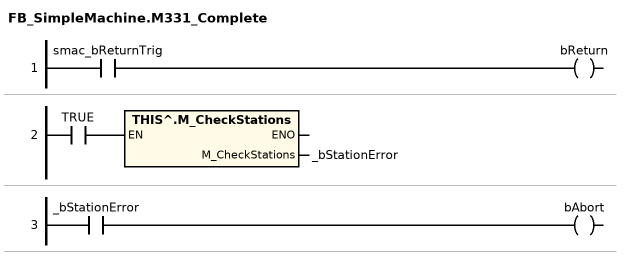
// NETWORK 1
bReturn := smac_bReturnTrig;

// NETWORK 2
_bStationError := THIS^.M_CheckStations();

// NETWORK 3
bAbort := _bStationError;
END_METHOD

(* In this state the most recent execution status should be maintained while
awaiting an explicit 'Unhold' command once internal conditions are satisfactory. *)
METHOD M411_Held : BOOL
VAR_OUTPUT
	(* This should be set to true if an explicit 'Unhold' command is received.
	Once set to true, the state machine will move to the 'Unholding' state. *)
	bUnhold	: BOOL;
	(* This should be set to true if an external source requests that the module
	exit its current state and come to a controlled stop. Once set to true, the
	state machine will move to the 'Stopping' state. *)
	bStop	: BOOL;
	(* This should be set to true if a potentially hazardous error or a safety
	fault has occurred in any tasks. Once set to true, the state machine will
	move to the 'Aborting' state. *)
	bAbort	: BOOL;
END_VAR
VAR
	_bStationError: BOOL;
END_VAR
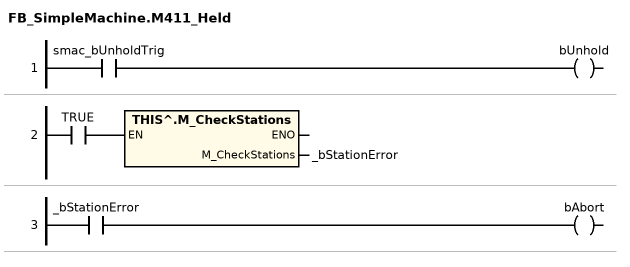
// NETWORK 1
bUnhold := smac_bUnholdTrig;

// NETWORK 2
_bStationError := THIS^.M_CheckStations();

// NETWORK 3
bAbort := _bStationError;
END_METHOD

(* In this state the most recent execution status should be maintained while
awaiting an explicit 'Unsuspend' command once external conditions are satisfactory. *)
METHOD M511_Suspended : BOOL
VAR_OUTPUT
	(* This should be set to true if an explicit 'Unsuspend' command is received.
	Once set to true, the state machine will move to the 'Unsuspending' state. *)
	bUnsuspend	: BOOL;
	(* This should be set to true if an external source requests that the module
	exit its current state and come to a controlled stop. Once set to true, the
	state machine will move to the 'Stopping' state. *)
	bStop	: BOOL;
	(* This should be set to true if a potentially hazardous error or a safety
	fault has occurred in any tasks. Once set to true, the state machine will
	move to the 'Aborting' state. *)
	bAbort	: BOOL;
END_VAR
VAR
	_bStationError: BOOL;
END_VAR
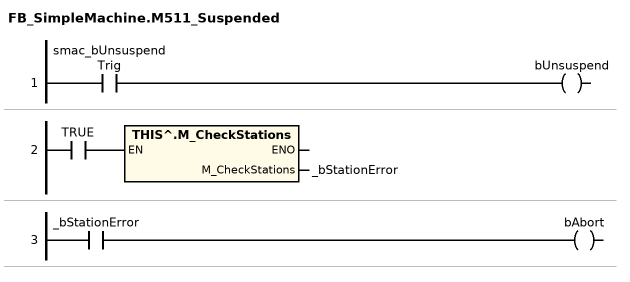
// NETWORK 1
bUnsuspend := smac_bUnsuspendTrig;

// NETWORK 2
_bStationError := THIS^.M_CheckStations();

// NETWORK 3
bAbort := _bStationError;
END_METHOD

END_FUNCTION_BLOCK

// Concrete/FB_StandardStation
FUNCTION_BLOCK FB_StandardStation EXTENDS FB_Station
VAR CONSTANT
	intMAX_USER_PROMPTS: INT := 255;
END_VAR
VAR_INPUT
	(* Station will start running process cycle once this is set to
		TRUE, and then will wait for this to be set to FALSE before
		resetting back to initial step. *)
	in_bRunCycleCommand: BOOL;
	(* Array of user prompts. *)
	in_arrUserPrompts: ARRAY[1..255] OF ST_Prompt;
	(* User retry signal for an exception state. *)
	in_bUserRetry: BOOL;
	(* User stop machine signal for an exception state. *)
	in_bUserAbort: BOOL;
END_VAR
VAR_OUTPUT
	(* Station should set this to TRUE while the process cycle is
		not running, and FALSE while running. *)
	out_bReadyToRun: BOOL;
	(* ID of the current user prompt. *)
	out_udintUserPromptCode: UDINT;
	(* Default message of the current user prompt. *)
	out_strUserPromptMessage: T_MaxString;
END_VAR
VAR
END_VAR

(* Sets ready to run to TRUE and waits for run cycle command to be reset. *)
METHOD M_AwaitCycleEnd : BOOL
VAR_INPUT
END_VAR
M_AwaitCycleEnd := FALSE;
IF NOT out_bReadyToRun THEN
	THIS^.M_LogMessage('Cycle complete.');
END_IF
out_bReadyToRun := TRUE;
IF NOT in_bRunCycleCommand THEN
	M_AwaitCycleEnd := TRUE;
END_IF
END_METHOD

(* Sets ready to run to TRUE and then waits for run cycle command. *)
METHOD M_AwaitCycleStart : BOOL
VAR_INPUT
END_VAR
M_AwaitCycleStart := FALSE;
out_bReadyToRun := TRUE;
IF in_bRunCycleCommand THEN
	out_bReadyToRun := FALSE;
	M_AwaitCycleStart := TRUE;
END_IF
END_METHOD

(* Clears the user prompt outputs. *)
METHOD M_ClearUserPrompt : BOOL
VAR_INPUT
END_VAR
out_strUserPromptMessage := '';
out_udintUserPromptCode := 0;
M_ClearUserPrompt := TRUE;
END_METHOD

(* Sets user prompt based on given code, and awaits user input. *)
METHOD M_HandleException : BOOL
VAR_INPUT
	(* Prompt code for the exception message. *)
	_in_udintPromptCode: UDINT;
	(* Error code to set in case user aborts. *)
	_in_udintErrorCode: UDINT;
END_VAR
VAR_OUTPUT
END_VAR
M_HandleException := FALSE;
THIS^.M_SetUserPrompt(_in_udintPromptCode);
IF in_bUserRetry THEN
	THIS^.M_ClearUserPrompt();
	M_HandleException := TRUE;
ELSIF in_bUserAbort THEN
	THIS^.M_SetError(_in_udintErrorCode, 'User chose to abort after an exception.');
END_IF
END_METHOD

METHOD M_ResetCycle : BOOL
VAR_INPUT
END_VAR
out_bReadyToRun := FALSE;
M_ResetCycle := TRUE;
END_METHOD

(* Sets out_strUserPromptCode and out_strUserPromptMessage based on
	the given user prompt code. *)
METHOD M_SetUserPrompt : BOOL
VAR_INPUT
	(* Prompt code to use for this user prompt. *)
	_in_udintCode: UDINT;
END_VAR

VAR
	_strMessage: T_MaxString;
	_intIndex: INT;
END_VAR
FOR _intIndex := 1 TO intMAX_USER_PROMPTS DO
	IF in_arrUserPrompts[_intIndex].udintCode = _in_udintCode THEN
		_strMessage := in_arrUserPrompts[_intIndex].strMessage;
		EXIT;
	END_IF
END_FOR
IF out_udintUserPromptCode <> _in_udintCode THEN
	IF LEN(_strMessage) > 0 THEN
		THIS^.M_LogMessage(_strMessage);
	ELSE
		THIS^.M_LogWarning('Prompt message not found!');
	END_IF
END_IF
out_strUserPromptMessage := _strMessage;
out_udintUserPromptCode := _in_udintCode;
M_SetUserPrompt := TRUE;
END_METHOD

END_FUNCTION_BLOCK

// Interfaces/State Machine/Stateful/I_ExecuteStateOnly
(* This interface only implements the methods for the Execute state. *)
INTERFACE I_ExecuteStateOnly EXTENDS I_SimpleExecuteStateOnly

(* Runs for a single cycle when entering the execute state. *)
METHOD M310_Execute_Entry : BOOL
VAR_INPUT
END_VAR
END_METHOD

(* Runs for a single cycle when exiting the execute state. *)
METHOD M312_Execute_Exit : BOOL
VAR_INPUT
END_VAR
END_METHOD

END_INTERFACE

// Interfaces/Stations/I_StationDeviceControl
INTERFACE I_StationDeviceControl

(* Aborts all devices set in the station. *)
METHOD M_AbortDevices : BOOL
VAR_INPUT
END_VAR
END_METHOD

(* Clears all devices set in the station. *)
METHOD M_ClearDevices : BOOL
VAR_INPUT
END_VAR
END_METHOD

(* Completes all devices set in the station. *)
METHOD M_CompleteDevices : BOOL
VAR_INPUT
END_VAR
END_METHOD

(* Holds all devices set in the station. *)
METHOD M_HoldDevices : BOOL
VAR_INPUT
END_VAR
END_METHOD

(* Resets all devices set in the station. *)
METHOD M_ResetDevices : BOOL
VAR_INPUT
END_VAR
END_METHOD

(* Starts all devices set in the station. *)
METHOD M_StartDevices : BOOL
VAR_INPUT
END_VAR
END_METHOD

(* Stops all devices set in the station. *)
METHOD M_StopDevices : BOOL
VAR_INPUT
END_VAR
END_METHOD

(* Suspends all devices set in the station. *)
METHOD M_SuspendDevices : BOOL
VAR_INPUT
END_VAR
END_METHOD

(* Unholds all devices set in the station. *)
METHOD M_UnholdDevices : BOOL
VAR_INPUT
END_VAR
END_METHOD

(* Unsuspends all devices set in the station. *)
METHOD M_UnsuspendDevices : BOOL
VAR_INPUT
END_VAR
END_METHOD

END_INTERFACE

// Project Information/F_GetCompany
// This function has been automatically generated from the project information.
{attribute 'signature_flag' := '1073741824'}
{attribute 'TcGenerated'}
{attribute 'no-analysis'}
FUNCTION F_GetCompany : WSTRING
VAR_INPUT
	
END_VAR

F_GetCompany := "Sensata Technologies";

END_FUNCTION

// Project Information/F_GetTitle
// This function has been automatically generated from the project information.
{attribute 'signature_flag' := '1073741824'}
{attribute 'TcGenerated'}
{attribute 'no-analysis'}
FUNCTION F_GetTitle : WSTRING
VAR_INPUT
	
END_VAR

F_GetTitle := "Sensata_Common";

END_FUNCTION

// Project Information/F_GetVersion
// This function has been automatically generated from the project information.
{attribute 'signature_flag' := '1073741824'}
{attribute 'TcGenerated'}
{attribute 'no-analysis'}
FUNCTION F_GetVersion : ST_LibVersion
VAR_INPUT
	
END_VAR

F_GetVersion.iMajor := 1;
F_GetVersion.iMinor := 0;
F_GetVersion.iBuild := 0;
F_GetVersion.iRevision := 0;

END_FUNCTION
